PROGRAM Vertical_Translation_Y2
VAR
//Outputs: Power for Limit switches, Home Sensors, etc.
    bFwdLimitPower AT %Q* : BOOL := TRUE;
    bBwdLimitPower AT %Q* : BOOL := TRUE;
    //bPowerSwitchesAxis1 AT %Q*: BOOL:= TRUE;

//Hardware interlocks
    //bInterlockFwdOK AT %I*: BOOL;
END_VAR

//Initial parameters of an Axis
(*IF _TaskInfo[fbGetCurTaskIndex.index].FirstCycle THEN
    //Initial default values:
    GVL.astAxes[1].stConfig.eHomeSeq := 0;
    GVL.astAxes[1].stConfig.fHomePosition := 0.0;
    GVL.astAxes[1].stConfig.fHomeFinishDistance := 0.0;
    GVL.astAxes[1].stConfig.eRestorePosition := E_RestorePosition.eRestoreWithoutHome;
END_IF*)

astAxes[AXIS_VERTICAL_TRANSLATION_Y2].stControl.bEnable := TRUE;
astAxes[AXIS_VERTICAL_TRANSLATION_Y2].stDescription.sAxisName := 'VERT_Y2';
//Define ACTIONS() or write exclusive code for an specific axis.
(*Eg. Stop when temperature reaches certain values, reduce speed if  a signal is activated, etc.
Eg. GVL.astAxes[x].stControl.bInterlockFwd := NOT bInterlockFwdOK;*)

END_PROGRAM

(* stored: Version 1.1.0.1, ProductVersion 3.1.4024.12
   POU Vertical_Translation_Y2: Id {3b7b9996-05d4-43b8-8768-65e5883d1014}, SpecialFunc None *)
